PROGRAM MAIN
VAR
	pmlbase : PML_StatePattern_Base;
	packmlmachine : PMLStateMachine;
	pmlmethod : PML_Method_Sample := (PackMLStateMachine := packmlmachine);
END_VAR

packmlmachine();
pmlmethod();

END_PROGRAM

(* stored: Version 1.1.0.1, ProductVersion 3.1.4024.12
   POU MAIN: Id {42a06358-885d-4ebb-8314-bfbbbdbdf83c}, SpecialFunc None *)
